PROGRAM task1
VAR
	PRG_Reis: INT;
	bReisGestart: BOOL;
END_VAR

// Start de reis
IF NOT bReisGestart THEN
    bReisGestart := TRUE;
    sStatusTekst := 'Ik ben onderweg naar Deventer...';
END_IF

// Aankomst in Deventer
IF bReisGestart AND NOT bInDeventer THEN
    bInDeventer := TRUE;
    sStatusTekst := 'Ik ben in Deventer. Ik wacht op koffie...';
END_IF

// Wachten op koffie van Task 2
IF bInDeventer AND bKoffieGereed THEN
    sStatusTekst := 'Koffie ontvangen! Ik reis door naar school.';
END_IF

END_PROGRAM

(* stored: Version 1.1.0.1, ProductVersion 3.1.4024.15
   POU task1: Id {dbff9976-da5b-4f60-8d50-96264a8bb7e1}, SpecialFunc None *)
